PROGRAM Axis9
VAR
	fbPower: MC_POWER;
	Axis: AXIS_REF;
	biLimFwd AT %I*: BOOL;
	biLimBwd AT %I*: BOOL;
	boBrake AT %Q*:BOOL;
	bEnable: BOOL := TRUE;
	rPosition AT %Q*:REAL;
	rVelocity AT %Q*:REAL;
	roPosition AT %Q*:REAL;
	fbReadActialPosition: MC_ReadActualPosition;
	fbHalt: MC_Halt;
	boHalt AT%Q*:BOOL;
	fbMoveAbsolute: MC_MoveAbsolute;
	boMoveAbsolute AT%Q*:BOOL;
	fbReadActualVelocity: MC_ReadActualVelocity;
END_VAR

fbPower(Axis:=Axis,
	Enable:=bEnable,
	Enable_Positive:=biLimFwd,
	Enable_Negative:=biLimBwd);
boBrake:=bEnable;
fbReadActialPosition(
	Axis:=Axis , 
	Enable:=TRUE , 
	Valid=> , 
	Busy=> , 
	Error=> , 
	ErrorID=> , 
	Position=>rPosition );
fbHalt(
	Axis:=Axis , 
	Execute:=boHalt , 
	Deceleration:= , 
	Jerk:= , 
	BufferMode:= , 
	Options:= , 
	Done=>, 
	Busy=> , 
	Active=> , 
	CommandAborted=> , 
	Error=> , 
	ErrorID=> );
fbMoveAbsolute(
	Axis:=Axis , 
	Execute:=boMoveAbsolute , 
	Position:=roPosition , 
	Velocity:=0.1 , 
	Acceleration:= , 
	Deceleration:= , 
	Jerk:= , 
	BufferMode:= , 
	Options:= , 
	Done=> , 
	Busy=> , 
	Active=> , 
	CommandAborted=> , 
	Error=> , 
	ErrorID=> );
fbReadActualVelocity(
	Axis:=Axis , 
	Enable:=TRUE , 
	Valid=> , 
	Busy=> , 
	Error=> , 
	ErrorID=> , 
	ActualVelocity=>rVelocity );

END_PROGRAM

(* stored: Version 1.1.0.1, ProductVersion 3.1.4022.3
   POU Axis9: Id {a1a742c9-0b68-41dc-add9-77d4a025f838}, SpecialFunc None *)
